{attribute 'qualified_only'}
VAR_GLOBAL CONSTANT
	Itf0			: Result := -2;
	Str0			: Result := -3;
	ItfEq			: Result := -4;
	NoMatch			: Result := -5;
	Ptr0			: Result := -6;
	InvRef			: Result := -7;
	Ovf				: Result := -8;
	Udf				: Result := -9;
	Idx				: Result := -10;
	TcLib			: Result := -11;
	InfLoop			: Result := -12;
END_VAR

(* stored: Version 1.1.0.1
   GVL Err: Id {6e918af6-d1f2-4bc6-828b-2f612da986e9} *)
